TYPE ST_MV_HD_Zustand :
STRUCT
	Kuehlung_Anford		: BOOL;
	Filterpumpe_Anford	: BOOL;
	Betrieb				: BOOL;

	Kommunikation		: BOOL;

	Stoerung				: BOOL;
	Stoerung_Code		: WORD;

	Warnung				: BOOL;
	Warnung_Code		: WORD;

	Status				: SINT;
END_STRUCT
END_TYPE

(* stored: Version 1.1.0.1, ProductVersion 3.1.4024.9
   DUT ST_MV_HD_Zustand: Id {30b1c64f-3464-40d2-b188-d922b21a1937} *)
